// SIMATIC S7-200 project (STEP 7-Micro/WIN), CPU 221 REL 01.10

SYMBOL_TABLE USER1
star             I0.0
tops             I0.1
den              Q0.0
END_SYMBOL_TABLE

ORGANIZATION_BLOCK MAIN:OB1
TITLE=PROGRAM COMMENTS
BEGIN
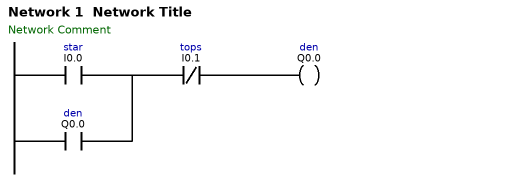
Network 1 // Network Title
// Network Comment
LD     star:I0.0
O      den:Q0.0
AN     tops:I0.1
=      den:Q0.0
END_ORGANIZATION_BLOCK
